{attribute 'qualified_only'}
VAR_GLOBAL
	{attribute 'OPC.UA.DA' := '1'}
    QrReader : ST_QrSkill;

    {attribute 'OPC.UA.DA' := '1'}
    RobotMove : ST_RobotMoveSkill;

    {attribute 'OPC.UA.DA' := '1'}
    Gripper : ST_GripperSkill;

END_VAR

(* stored: Version 1.1.0.1, ProductVersion 3.1.4026.18
   GVL OPCUA: Id {81992575-26c5-4473-91f9-1a7612771094} *)
